(* IEC 61131-3 sources: AXOpen/src/components.cognex.vision/ctrl/src/AxoInsight/v_24_0_0/TypeStructuresAndEnums, 17 files *)

(* ---- AxoInsight_AcquisitionControl.st ---- *)
NAMESPACE AXOpen.Components.Cognex.Vision.v_24_0_0
    TYPE
        {#ix-attr:[Container(Layout.Wrap)]}
        {S7.extern=ReadWrite}
        AxoInsight_AcquisitionControl :
        STRUCT
            {#ix-set:AttributeName = "<#Trigger enable#>"}
            TriggerEnable 			:	BOOL;
            {#ix-set:AttributeName = "<#Trigger#>"}
            Trigger					:	BOOL;
            {#ix-set:AttributeName = "<#Clear exposure complete#>"}
            ClearExposureComplete :  BOOL;
            {#ix-set:AttributeName = "<#Set offline#>"}
            SetOffline :  BOOL;
        END_STRUCT;
    END_TYPE
END_NAMESPACE

(* ---- AxoInsight_AcquisitionStatus.st ---- *)
NAMESPACE AXOpen.Components.Cognex.Vision.v_24_0_0
    TYPE
        {#ix-attr:[Container(Layout.Wrap)]}
        {S7.extern=ReadWrite}
        AxoInsight_AcquisitionStatus :
        STRUCT
            {#ix-set:AttributeName = "<#Trigger ready#>"}
            TriggerReady 		:	BOOL;
            {#ix-set:AttributeName = "<#Trigger acknowledge#>"}
            TriggerAcknowledge 	:	BOOL;
            {#ix-set:AttributeName = "<#Exposure complete#>"}
            ExposureComplete	:	BOOL;
            {#ix-set:AttributeName = "<#Missed acquisition#>"}
            MissedAcquisition 	:	BOOL;
            {#ix-set:AttributeName = "<#Offline reason 0#>"}
            OfflineReason0      :   BOOL;
            {#ix-set:AttributeName = "<#Offline reason 1#>"}
            OfflineReason1      :   BOOL;
            {#ix-set:AttributeName = "<#Offline reason 2#>"}
            OfflineReason2      :   BOOL;
            {#ix-set:AttributeName = "<#Online#>"}
            Online              :   BOOL;
            {#ix-set:AttributeName = "<#Acquisition ID#>"}
            AcquisitionID       :   UINT;
        END_STRUCT;
    END_TYPE
END_NAMESPACE

(* ---- AxoInsight_CommandControl.st ---- *)
NAMESPACE AXOpen.Components.Cognex.Vision.v_24_0_0
    TYPE
        {#ix-attr:[Container(Layout.Wrap)]}
        {S7.extern=ReadWrite}
        AxoInsight_CommandControl :
        STRUCT
            {#ix-set:AttributeName = "<#Command#>"}
            Command        : UINT;
        END_STRUCT;
    END_TYPE
END_NAMESPACE

(* ---- AxoInsight_CommandStatus.st ---- *)
NAMESPACE AXOpen.Components.Cognex.Vision.v_24_0_0
    TYPE
        {#ix-attr:[Container(Layout.Wrap)]}
        {S7.extern=ReadWrite}
        AxoInsight_CommandStatus :
        STRUCT
            {#ix-set:AttributeName = "<#Current job ID#>"}
            CurrentJobID  : UINT;
        END_STRUCT;
    END_TYPE
END_NAMESPACE

(* ---- AxoInsight_Config.st ---- *)
NAMESPACE AXOpen.Components.Cognex.Vision.v_24_0_0
    TYPE
        {#ix-attr:[Container(Layout.Wrap)]}
        {S7.extern=ReadWrite}
        AxoInsight_Config :
        STRUCT
            {#ix-set:AttributeName = "<#Info time#>"}
            InfoTime : LTIME := LT#10S;
            {#ix-set:AttributeName = "<#Error time#>"}
            ErrorTime : LTIME := LT#50S;
            {#ix-set:AttributeName = "<#Max job number#>"}
            MaxJobNumber : UINT := UINT#999;
            {#ix-set:AttributeName = "<#Result data size#>"}
            ResultDataSize : UINT;
            {#ix-set:AttributeName = "<#User data size#>"}
            UserDataSize : UINT;
            {#ix-set:AttributeName = "<#Hardware IDs#>"}
            HWIDs : AxoInsight_HWIDs;
        END_STRUCT;
    END_TYPE
END_NAMESPACE

(* ---- AxoInsight_InspectionControl.st ---- *)
NAMESPACE AXOpen.Components.Cognex.Vision.v_24_0_0
    TYPE
        {#ix-attr:[Container(Layout.Wrap)]}
        {S7.extern=ReadWrite}
        AxoInsight_InspectionControl :
        STRUCT
            {#ix-set:AttributeName = "<#Enable results buffering#>"}
            EnableResultsBuffering          :   BOOL;
            {#ix-set:AttributeName = "<#Acknowledge inspection results#>"}
            AcknowledgeInspectionResults    :   BOOL;
            {#ix-set:AttributeName = "<#Extended user data set#>"}
            ExtendedUserDataSet             :   BOOL;
            {#ix-set:AttributeName = "<#Execute command#>"}
            ExecuteCommand                  :   BOOL;
            {#ix-set:AttributeName = "<#Clear error#>"}
            ClearError                      :   BOOL;
        END_STRUCT;
    END_TYPE
END_NAMESPACE

(* ---- AxoInsight_InspectionStatus.st ---- *)
NAMESPACE AXOpen.Components.Cognex.Vision.v_24_0_0
    TYPE
        {#ix-attr:[Container(Layout.Wrap)]}
        {S7.extern=ReadWrite}
        AxoInsight_InspectionStatus :
        STRUCT
            {#ix-set:AttributeName = "<#System busy#>"}
            SystemBusy                      :   BOOL;
            {#ix-set:AttributeName = "<#Inspection completed#>"}
            InspectionCompleted             :   BOOL;
            {#ix-set:AttributeName = "<#Results buffer overrun#>"}
            ResultsBufferOverrun            :   BOOL;
            {#ix-set:AttributeName = "<#Results valid#>"}
            ResultsValid                    :   BOOL;
            {#ix-set:AttributeName = "<#Command executing#>"}
            CommandExecuting                :   BOOL;
            {#ix-set:AttributeName = "<#Command complete#>"}
            CommandComplete                 :   BOOL;
            {#ix-set:AttributeName = "<#Command failed#>"}
            CommandFailed                   :   BOOL;
            {#ix-set:AttributeName = "<#Extended user data set acknowledge#>"}
            ExtendedUserDataSetAcknowledge  :   BOOL;
            {#ix-set:AttributeName = "<#Overall job pass fail#>"}
            OverallJobPassFail              :   BOOL;
            {#ix-set:AttributeName = "<#Test run ready#>"}
            TestRunReady                    :   BOOL;
            {#ix-set:AttributeName = "<#Error#>"}
            Error                           :   BOOL;
            {#ix-set:AttributeName = "<#Error code#>"}
            ErrorCode                       :   UINT;
        END_STRUCT;
    END_TYPE
END_NAMESPACE

(* ---- AxoInsight_Results.st ---- *)
NAMESPACE AXOpen.Components.Cognex.Vision.v_24_0_0
    TYPE
        {#ix-attr:[Container(Layout.Wrap)]}
        {S7.extern=ReadWrite}
        AxoInsight_Results :
        STRUCT
            {#ix-set:AttributeName = "<#Inspection ID#>"}
            InspectionID : UINT;
            {#ix-set:AttributeName = "<#Result code#>"}
            ResultCode : UINT;
        END_STRUCT;
    END_TYPE
END_NAMESPACE

(* ---- AxoInsight_SoftEventControl.st ---- *)
NAMESPACE AXOpen.Components.Cognex.Vision.v_24_0_0
    TYPE
        {#ix-attr:[Container(Layout.Wrap)]}
        {S7.extern=ReadWrite}
        AxoInsight_SoftEventControl :
        STRUCT
            {#ix-set:AttributeName = "<#Trigger soft-event#>"}
            TriggerSoftEvent : AxoBoolArray8;
        END_STRUCT;
    END_TYPE
END_NAMESPACE

(* ---- AxoInsight_SoftEventStatus.st ---- *)
NAMESPACE AXOpen.Components.Cognex.Vision.v_24_0_0
    TYPE
        {#ix-attr:[Container(Layout.Wrap)]}
        {S7.extern=ReadWrite}
        AxoInsight_SoftEventStatus :
        STRUCT
            {#ix-set:AttributeName = "<#Trigger soft-event acknowledge#>"}
            TriggerSoftEventAcknowledge : AxoBoolArray8;
        END_STRUCT;
    END_TYPE
END_NAMESPACE

(* ---- eAxoInsight_ResultDataSize.st ---- *)
NAMESPACE AXOpen.Components.Cognex.Vision.v_24_0_0
    TYPE PUBLIC
        eAxoInsight_ResultDataSize : INT
        (
            RESULT_DATA_SIZE_INVALID := 0,
            RESULT_DATA_16B := 16,
            RESULT_DATA_32B := 32,
            RESULT_DATA_64B := 64,
            RESULT_DATA_128B := 128,
            RESULT_DATA_250B := 250
         ) := RESULT_DATA_64B;
    END_TYPE
END_NAMESPACE

(* ---- eAxoInsight_UserDataSize.st ---- *)
NAMESPACE AXOpen.Components.Cognex.Vision.v_24_0_0
    TYPE PUBLIC
        eAxoInsight_UserDataSize : INT
        (
            USER_DATA_SIZE_INVALID := 0,
            USER_DATA_16B := 16,
            USER_DATA_32B := 32,
            USER_DATA_64B := 64,
            USER_DATA_128B := 128,
            USER_DATA_254B := 254
         ) := USER_DATA_64B;
    END_TYPE
END_NAMESPACE

(* ---- AxoBoolArray8.st ---- *)
NAMESPACE AXOpen.Components.Cognex.Vision.v_24_0_0
    {S7.extern=ReadWrite}
    CLASS PUBLIC AxoBoolArray8 EXTENDS AXOpen.Core.AxoBoolArray
        VAR PUBLIC
            Data : ARRAY [0..7] OF BOOL;
        END_VAR
    END_CLASS
END_NAMESPACE

(* ---- AxoInsight_HWIDs.st ---- *)
NAMESPACE AXOpen.Components.Cognex.Vision.v_24_0_0
   {S7.extern=ReadWrite}
	CLASS AxoInsight_HWIDs
      VAR PUBLIC
         {#ix-set:AttributeName = "<#Hardware ID of the device#>"}
         HW_Device              : UINT;
         {#ix-set:AttributeName = "<#Hardware ID 'AcquisitionControl' submodule#>"}
         HW_AcquisitionControl     : UINT;
         {#ix-set:AttributeName = "<#Hardware ID 'AcquisitionStatus' submodule#>"}
         HW_AcquisitionStatus   : UINT;
         {#ix-set:AttributeName = "<#Hardware ID 'InspectionControl' submodule#>"}
         HW_InspectionControl   : UINT;
         {#ix-set:AttributeName = "<#Hardware ID 'InspectionStatus' submodule#>"}
         HW_InspectionStatus   : UINT;
         {#ix-set:AttributeName = "<#Hardware ID 'CommandControl' submodule#>"}
         HW_CommandControl   : UINT;
         {#ix-set:AttributeName = "<#Hardware ID 'SoftEventControl' submodule#>"}
         HW_SoftEventControl   : UINT;
         {#ix-set:AttributeName = "<#Hardware ID 'UserDataSlot_7' submodule#>"}
         HW_UserDataSlot_7   : UINT;
         {#ix-set:AttributeName = "<#Hardware ID 'UserDataSlot_8' submodule#>"}
         HW_UserDataSlot_8   : UINT;
         {#ix-set:AttributeName = "<#Hardware ID 'UserDataSlot_9' submodule#>"}
         HW_UserDataSlot_9   : UINT;
         {#ix-set:AttributeName = "<#Hardware ID 'UserDataSlot_10' submodule#>"}
         HW_UserDataSlot_10   : UINT;
         {#ix-set:AttributeName = "<#Hardware ID 'ResultData_Slot_11' submodule#>"}
         HW_ResultData_Slot_11    : UINT;
         {#ix-set:AttributeName = "<#Hardware ID 'ResultData_Slot_12' submodule#>"}
         HW_ResultData_Slot_12    : UINT;
         {#ix-set:AttributeName = "<#Hardware ID 'ResultData_Slot_13' submodule#>"}
         HW_ResultData_Slot_13    : UINT;
         {#ix-set:AttributeName = "<#Hardware ID 'ResultData_Slot_14' submodule#>"}
         HW_ResultData_Slot_14    : UINT;
      END_VAR
   END_CLASS
END_NAMESPACE

(* ---- AxoInsight_ResultData.st ---- *)
NAMESPACE AXOpen.Components.Cognex.Vision.v_24_0_0
    {S7.extern=ReadWrite}
    CLASS PUBLIC AxoInsight_ResultData EXTENDS AXOpen.Core.AxoByteArray
        VAR PUBLIC
            Data : ARRAY [0..999] OF BYTE;
        END_VAR
    END_CLASS
END_NAMESPACE

(* ---- AxoInsight_Status.st ---- *)
USING AXOpen.Core;
NAMESPACE AXOpen.Components.Cognex.Vision.v_24_0_0
    {#ix-attr:[Container(Layout.Stack)]}
    {S7.extern=ReadWrite}
    CLASS AxoInsight_Status EXTENDS AXOpen.Components.Abstractions.AxoComponent_Status
        VAR PUBLIC
            {#ix-attr:[Container(Layout.Wrap)]}
            {#ix-set:AttributeName = "<#Current job name#>"}
            CurrentJobName : STRING;
            {#ix-set:AttributeName = "<#Current job number#>"}
            CurrentJobNumber : UINT;
        END_VAR
    END_CLASS
END_NAMESPACE

(* ---- AxoInsight_UserData.st ---- *)
NAMESPACE AXOpen.Components.Cognex.Vision.v_24_0_0
    {S7.extern=ReadWrite}
    CLASS PUBLIC AxoInsight_UserData EXTENDS AXOpen.Core.AxoByteArray
        VAR PUBLIC
            Data : ARRAY [0..255] OF BYTE;
        END_VAR
    END_CLASS
END_NAMESPACE
